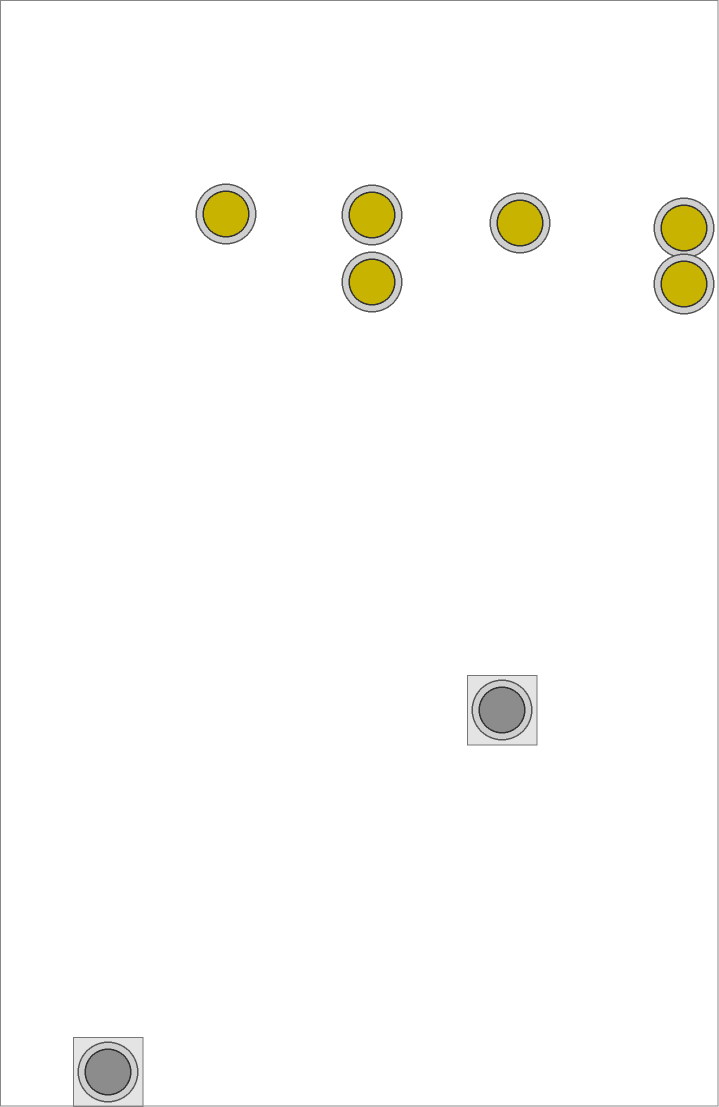
VISUALIZATION Screen1  // 719x1107
    Lamp1 (191,179 70x70), variable: HMI.led1_1, style: Lamp-Lamp1-Yellow
    Lamp1 (337,247 70x70), variable: HMI.led2_2, style: Lamp-Lamp1-Yellow
    Lamp1 (337,180 70x70), variable: HMI.led2_1, style: Lamp-Lamp1-Yellow
    Lamp1 (485,188 70x70), variable: HMI.led3, style: Lamp-Lamp1-Yellow
    Lamp1 (649,193 70x70), variable: HMI.led4_1, style: Lamp-Lamp1-Yellow
    Lamp1 (649,249 70x70), variable: HMI.led4_2, style: Lamp-Lamp1-Yellow
    PushSwitch (467,675 70x70), variable: HMI.btn, behaviour: TAP, style: Switch-PushSwitch-Gray
    PushSwitch (73,1037 70x70), variable: MAIN.isDay, behaviour: TOGGLE, style: Switch-PushSwitch-Gray
END_VISUALIZATION

(* stored: Version 1.1.0.1, ProductVersion 3.1.4024.12
   Visu Screen1: Id {6923abbf-1f3c-4bab-890b-3470c7d8ab97} *)
